METHOD AddIBufferFullChilds
VAR_INPUT
	pFB_ChildTypeIBuffer: POINTER TO FB_IBuffer;
END_VAR
// Method add childs with BufferFull information to the array
IF (usiNumOfIBufferFullChild <= (Base_Const.cMaxNrOfChilds-1)) THEN
	// Add child controller to list
	a_IBufferFullChildCtrl[usiNumOfIBufferFullChild] := pFB_ChildTypeIBuffer^;

	// Inc. number of IBufferFull childs
	usiNumOfIBufferFullChild:= usiNumOfIBufferFullChild+1;
END_IF
END_METHOD

METHOD AddSeqChild
VAR_INPUT
	stSequence: T_Sequence;
END_VAR
// Method add a sequence to list
IF (usiNumOfSeq <= (Base_Const.cMaxNrOfChilds-1)) THEN
	aListOfSeq[usiNumOfSeq].pChild:= stSequence.pChild;
	aListOfSeq[usiNumOfSeq].uinGroupRun:= stSequence.uinGroupRun;
	aListOfSeq[usiNumOfSeq].uinGroupStop:= stSequence.uinGroupStop;
	aListOfSeq[usiNumOfSeq].intCmdSeqRun:= stSequence.intCmdSeqRun;
	aListOfSeq[usiNumOfSeq].intStatusSeqRun:= stSequence.intStatusSeqRun;
	aListOfSeq[usiNumOfSeq].intStatusSeqRun2:= stSequence.intStatusSeqRun2;
	aListOfSeq[usiNumOfSeq].intCmdSeqStop:= stSequence.intCmdSeqStop;
	aListOfSeq[usiNumOfSeq].intStatusSeqStop:= stSequence.intStatusSeqStop;
	// Inc. number of sequence
	usiNumOfSeq:= usiNumOfSeq+1;
	// Check if the pointer is valid
	IF (stSequence.pChild<>0) THEN
		usiNumOfValidPointerSeqChild:= usiNumOfValidPointerSeqChild+1;
	END_IF
END_IF
END_METHOD

METHOD PROTECTED Always : BOOL
SUPER^.Always();

// ---------------------------------------------------------------------------------
// Simulation
IF (CIf.SwCfg.bolSimulation) THEN
	SIf_Cur^.bolKeepAliveHost := NOT SIf_Cur^.bolKeepAlivePlc;
	// Simulate inputs from global module for general supervision (no physical inputs)
	SIf_In^.bolEmoOk.intern := TRUE;
	SIf_In^.bolReady.intern := TRUE;
END_IF

// ----------------------------------------------------------------------------------
// cyclic actions outside of statemachine
IF (me.StateMachine.intState<>cSTA_SINGLE_ANSWER) THEN
	
	// Ready Output
	SIf_Out^.bolReady.intern := (me.StateMachine.intState = BASE_PLC.cSTA_RUN) AND (me.Alarm.eActivAlmClass < BASE_PLC.E_AlmClass.TSTOP);
	
	// Emergency Off
	IF ((SIf_In^.bolEmoOk.intern = FALSE) AND (me.StateMachine.intState <> cSTA_EOFF) AND (me.StateMachine.intState <> cSTA_EOFFBusy)
		AND (me.StateMachine.intState <> cSTA_ERROR) AND (me.StateMachine.intState <> cSTA_ERRORQuit)) THEN
		me.StateMachine.intStateNext := cSTA_EOFFBusy;				
	END_IF
	
	// As long as EMO is not OK, set Alarm
	IF (SIf_In^.bolEmoOk.intern = FALSE) AND ((me.StateMachine.intState = cSTA_EOFF) OR (me.StateMachine.intState = cSTA_EOFFBusy)) THEN
		//SIf_MOD.Alm[E_ALM_MOD.EmergencyOff].strText := 'Emergency off active';
		pfbAlarmCtrl^.setAlarm(CIf.Info.intCtrlId,E_ALM_MOD.EmergencyOff,0,ADR(SIf_MOD.Alm),E_AlmState.RST,CIf.Job.eMe_ActivAlmClass);
	END_IF
	
END_IF

//-------------------------------------------------------------------------------
// Keep Alive function to line controller with togglebit
//-------------------------------------------------------------------------------

// Communication to line control enabled
IF (SIf_Cfg^.bolComToLineControlEnabled = TRUE) THEN
	IF (SIf_Cur^.bolKeepAliveHost <> SIf_Cur^.bolKeepAlivePlc) THEN
		udinTimeToggle_ms := 0;
		SIf_Cur^.bolKeepAlivePlc := SIf_Cur^.bolKeepAliveHost;
	ELSE
		IF (udinTimeToggle_ms >= SIf_Par^.udiComTimeOutLineCtrl_ms) THEN
			//SIf_MOD.Alm[E_ALM_MOD.CommunicationError].strText := 'Communication error to line control'; 
			pfbAlarmCtrl^.setAlarm(CIf.Info.intCtrlId,E_ALM_MOD.CommunicationError,UDINT_TO_DINT(udinTimeToggle_ms),ADR(SIf_MOD.Alm),E_AlmState.RST,CIf.Job.eMe_ActivAlmClass);	
			me.StateMachine.intStateNext := cSTA_Error;	
		END_IF
		udinTimeToggle_ms:= udinTimeToggle_ms + me.FUBInfo.udiSample_ms;
	END_IF
// Communication to line control disabled
ELSE
	SIf_Cur^.bolKeepAliveHost:= NOT SIf_Cur^.bolKeepAlivePlc;
END_IF

//-------------------------------------------------------------------------------
// Calculate the sum of all items in the system and the capacity of the system
//-------------------------------------------------------------------------------
IF (usiNumOfIBufferChild>0) THEN 
	SIf_Cur^.dinNumOfItems:= 0;
	SIf_Cur^.dinMaxCapacity:= 0;
	FOR ii:= 0 TO (usiNumOfIBufferChild-1) DO
		SIf_Cur^.dinNumOfItems:= SIf_Cur^.dinNumOfItems + a_IBufferChildCtrl[ii].NumOfItems;
		SIf_Cur^.dinMaxCapacity:= SIf_Cur^.dinMaxCapacity + a_IBufferChildCtrl[ii].MaxCapacity;
	END_FOR
END_IF

//-------------------------------------------------------------------------------
// Write BufferFull for LineControl into SIF
//-------------------------------------------------------------------------------
IF (usiNumOfIBufferFullChild>0) THEN 
	FOR ii:= 0 TO (usiNumOfIBufferFullChild-1) DO
		SIf_Cur^.a_bBufferIsFull[ii]:= a_IBufferFullChildCtrl[ii].BufferFull;
	END_FOR
END_IF


// ----------------------------------------------------------------------------------
// Conditions Always

// EOFF exist in FB_CtrlModule. Not overrule.
(*
// overrule error always from base -> no EOFF State!! in EOFF go to OFF
IF (me.StateMachine.intStateNext = cSTA_EOFFBusy) THEN
	IF (me.StateMachine.intState=cSTA_OFF) THEN
		me.StateMachine.intStateNext := cSTA_OFF;
	ELSE // stay in OFF
		me.StateMachine.intStateNext := cSTA_OFFBusy;
	END_IF
*)
IF (me.Alarm.eActivAlmClass=E_AlmClass.STOP) AND (me.StateMachine.intStateNext<>cSTA_Error)
		AND ((me.StateMachine.intState = cSTA_RUN) OR (me.StateMachine.intState = cSTA_RUNBusy))THEN
	// alarm evt STOP
	me.StateMachine.intStateNext := cSTA_STOPBusy;	
END_IF
END_METHOD

{attribute 'object_name' := 'CheckAllChildStateOr'}
METHOD PROTECTED CheckAllChildStateOr : BOOL
VAR_INPUT
	In_intCheckState1: INT;
	In_intCheckState2: INT;
END_VAR
VAR
	uinIdx: UINT;
END_VAR
// check if all child controller have reached one of the two In_intCheckState
CheckAllChildStateOr := TRUE;
IF (CIf.Info.uinChildNbr > 0) THEN
	FOR uinIdx := 0 TO CIf.Info.uinChildNbr - 1 DO
		CheckAllChildStateOr := CheckAllChildStateOr AND ((CIf.Info.p_aCIf[uinIdx]^.Job.intState = In_intCheckState1) OR (CIf.Info.p_aCIf[uinIdx]^.Job.intState = In_intCheckState2));
		IF (CheckAllChildStateOr=FALSE) THEN	// at least one child has not whished state reached
			EXIT ;
		END_IF 
	END_FOR
END_IF
END_METHOD

METHOD checkChildAlmClass : BOOL
//------------------------------------------------------------------------------------------------------
// check child alarm classes
// set me alarm class active if at least one child has an EOFF
IF CheckAllChildAlmClass(E_AlmClass.EOFF) THEN
	CIf.Job.eMe_ActivAlmClass := E_AlmClass.EOFF;
	me.Alarm.bolfp := TRUE;
ELSIF CheckAllChildAlmClass(E_AlmClass.OFF) THEN
	CIf.Job.eMe_ActivAlmClass := E_AlmClass.OFF;
	me.Alarm.bolfp := TRUE;
ELSIF CheckAllChildAlmClass(E_AlmClass.STOP) THEN
	CIf.Job.eMe_ActivAlmClass := E_AlmClass.STOP;
	me.Alarm.bolfp := TRUE;
ELSIF CheckAllChildAlmClass(E_AlmClass.TSTOP) THEN
	CIf.Job.eMe_ActivAlmClass := E_AlmClass.TSTOP;
	me.Alarm.bolfp := TRUE;
ELSE
	IF (me.Alarm.bolfp) THEN
		CIf.Job.eMe_ActivAlmClass := E_AlmClass.NONE; // no reset necessary
		me.Alarm.bolfp := FALSE;
	END_IF
END_IF

//------------------------------------------------------------------------------------------------------
// set alarm class parent of childs
//------------------------------------------------------------------------------------------------------
// set alarm class parent of childs in the case of a parent EOFF or me=OFF or EOFF
IF (CIf.Job.eParent_ActivAlmClass=E_AlmClass.EOFF) THEN
	SetAllChildAlmClass(CIf.Job.eParent_ActivAlmClass);
ELSIF(CIf.Job.eMe_ActivAlmClass=E_AlmClass.EOFF) OR (CIf.Job.eMe_ActivAlmClass=E_AlmClass.OFF) THEN
	SetAllChildAlmClass(CIf.Job.eMe_ActivAlmClass);
ELSE
	// no important alarm for child active
	SetAllChildAlmClass(E_AlmClass.NONE);
END_IF
END_METHOD

METHOD PROTECTED checkValidPointer : BOOL
IF (usiNumOfSeq = usiNumOfValidPointerSeqChild) AND (SIf_Cfg<>0) AND (SIf_Par<>0) AND (SIf_Cur<>0) AND (SIf_In<>0) THEN
	checkValidPointer:= TRUE;
ELSE
	// Invalid child pointer
	checkValidPointer:= FALSE;	
	//SIf_MOD.Alm[E_ALM_MOD.InvalidPointer].strText := 'Invalid pointer';
	pfbAlarmCtrl^.setAlarm(CIf.Info.intCtrlId,E_ALM_MOD.InvalidPointer,0,ADR(SIf_MOD.Alm),E_AlmState.RST,CIf.Job.eMe_ActivAlmClass);	
END_IF
END_METHOD

METHOD PUBLIC CtrlInit : BOOL
VAR
	ii: INT;
END_VAR
SUPER^.CtrlInit();

// Initialize all child controller
// Childs are listed in list of sequences
FOR ii:=0 TO usiNumOfSeq-1 BY 1 DO	
	aListOfSeq[ii].pCIF := THIS^.AddChild(aListOfSeq[ii].pChild^);
END_FOR
END_METHOD

METHOD FB_init : BOOL
VAR_INPUT
	///if TRUE, the retain variables are initialized (warm start / cold start)
	bInitRetains: BOOL;
	///if TRUE, the instance afterwards gets moved into the copy code (online change)
	bInCopyCode: BOOL;
END_VAR
VAR
	ii: UINT;
END_VAR
// to manually change in new FUB implementation!!!
// define valid commands for this controller
FOR ii:= 0 TO (SIZEOF(CIf.Job.aCmdList)/SIZEOF(CIf.Job.aCmdList[0])-1) BY 1 DO
	IF (CIf.Job.aCmdList[ii].intCmd=cCMD_INITIALIZED) THEN
		// found first empty array element
		EXIT;
	END_IF
END_FOR

CIf.Job.aCmdList[ii].intCmd := cCMD_RUN;
CIf.Job.aCmdList[ii].strName := 'Run'; 
CIf.Job.aCmdList[ii].bolAvailable := TRUE;
ii := ii +1;
CIf.Job.aCmdList[ii].intCmd := cCMD_STOP;
CIf.Job.aCmdList[ii].strName := 'Stop'; 
CIf.Job.aCmdList[ii].bolAvailable := TRUE;
ii := ii +1;
CIf.Job.aCmdList[ii].intCmd := cCMD_STANDBY;
CIf.Job.aCmdList[ii].strName := 'Standby'; 
CIf.Job.aCmdList[ii].bolAvailable := TRUE;
ii := ii +1;

// set name of class/typ
CIf.Info.strType := 'FB_CtrlModule';
CIf.Info.strFullName := 'Base Controller Module';

// set alarm class
SIf_MOD.Alm[E_ALM_MOD.InvalidPointer].eAlmClass := E_AlmClass.STOP;
SIf_MOD.Alm[E_ALM_MOD.InvalidPointer].strText := 'Invalid pointer';
SIf_MOD.Alm[E_ALM_MOD.CommunicationError].eAlmClass := E_AlmClass.OFF;
SIf_MOD.Alm[E_ALM_MOD.CommunicationError].strText := 'Communication error to line control';
SIf_MOD.Alm[E_ALM_MOD.EmergencyOff].eAlmClass := E_AlmClass.EOFF;
SIf_MOD.Alm[E_ALM_MOD.EmergencyOff].strText := 'Emergency off active';
SIf_MOD.Alm[E_ALM_MOD.TimeoutStartGroup].eAlmClass := E_AlmClass.OFF;
SIf_MOD.Alm[E_ALM_MOD.TimeoutStartGroup].strText := 'Timeout start group';
SIf_MOD.Alm[E_ALM_MOD.TimeoutStopGroup].eAlmClass := E_AlmClass.OFF;
SIf_MOD.Alm[E_ALM_MOD.TimeoutStopGroup].strText := 'Timeout stop group';
SIf_MOD.Alm[E_ALM_MOD.NextModuleNotReadyWarning].eAlmClass := E_AlmClass.WARNING;
SIf_MOD.Alm[E_ALM_MOD.NextModuleNotReadyWarning].strText := 'Next Module is not Ready';
SIf_MOD.Alm[E_ALM_MOD.NextModuleNotReadyStop].eAlmClass := E_AlmClass.STOP;
SIf_MOD.Alm[E_ALM_MOD.NextModuleNotReadyStop].strText := 'Next Module is not Ready';

//*******************************************************************************
// initial values
//*******************************************************************************
udinTimeToggle_ms := 0;
// software configuration
CIf.SwCfg.bolExist := TRUE;
CIf.SwCfg.bolSimulation := FALSE;
me.AlarmConfig.bolChildrenAlarmPropagation := FALSE;

// No initialization for cfg and par in this base module!
// Pointer address of the property is not defined at this time
END_METHOD

METHOD PROTECTED FurtherReactions : BOOL
IF (	(NOT me.AlarmConfig.bolOffAlarmTransitionDisable)	AND (me.Alarm.eActivAlmClass=E_AlmClass.STOP)
	AND (me.StateMachine.intState<>cSTA_ERROR)				AND	(me.StateMachine.intState<>cSTA_ERRORQuit)
	AND	(me.StateMachine.intState<>cSTA_EOFF)				AND	(me.StateMachine.intState<>cSTA_EOFFBusy)
	AND	(me.StateMachine.intState<>cSTA_OFF)				AND	(me.StateMachine.intState<>cSTA_OFFBusy)
	AND (me.StateMachine.intState<>cSTA_STOP)				AND (me.StateMachine.intState<>cSTA_STOPBusy)
	AND	(me.StateMachine.intState>cSTA_PON)) THEN
	
	me.StateMachine.intStateNext := cSTA_STOPBusy;
	me.StateMachine.intState := cSTA_DONE;
	
ELSIF (	(NOT me.AlarmConfig.bolOffAlarmTransitionDisable)	AND (me.Alarm.eActivAlmClass=E_AlmClass.TSTOP)
	AND (me.StateMachine.intState<>cSTA_ERROR)				AND	(me.StateMachine.intState<>cSTA_ERRORQuit)
	AND	(me.StateMachine.intState<>cSTA_EOFF)				AND	(me.StateMachine.intState<>cSTA_EOFFBusy)
	AND	(me.StateMachine.intState<>cSTA_OFF)				AND	(me.StateMachine.intState<>cSTA_OFFBusy)
	AND (me.StateMachine.intState<>cSTA_STOP)				AND (me.StateMachine.intState<>cSTA_STOPBusy)
	AND	(me.StateMachine.intState>cSTA_PON)) THEN
	
	me.StateMachine.intStateNext := cSTA_STOPBusy;
	me.StateMachine.intState := cSTA_DONE;
	
END_IF
END_METHOD

METHOD PROTECTED getCmdState : STRING
VAR_INPUT
	intCmdState: INT;
	bolState: BOOL;
END_VAR
getCmdState := SUPER^.getCmdState(intCmdState:=intCmdState,bolState:=bolState); // get global/base defined cmds/states
IF (getCmdState='') THEN // global not defined get local
	// get string cmd/state string information in runtime
	IF (bolState=FALSE) THEN
		// cmd's
		CASE intCmdState OF
			cCMD_STANDBY: 
				getCmdState := 'cCMD_STANDBY';
		END_CASE
	ELSE
		// states
		CASE intCmdState OF	
			cSTA_STANDBY:
				getCmdState := 'cSTA_STANDBY';
			cSTA_STANDBYBusy:
				getCmdState := 'cSTA_STANDBYBusy';
			// SUB States
			cSTA_SUB_INITIALIZED:
				getCmdState := 'cSTA_SUB_INITIALIZED';
			cSTA_SUB_SEND_GROUP_CMD:
				getCmdState := 'cSTA_SUB_SEND_GROUP_CMD';
			cSTA_SUB_CHECK_GROUP_STATUS:
				getCmdState := 'cSTA_SUB_CHECK_GROUP_STATUS';
			cSTA_SUB_WAIT:
				getCmdState := 'cSTA_SUB_WAIT';
			cSTA_SUB_FINISHED:
				getCmdState := 'cSTA_SUB_FINISHED';
		END_CASE;
	END_IF
END_IF
END_METHOD

METHOD PROTECTED IoInBridge : BOOL
// digitale and analoge inputs read from hardware or forcing
SIf_In^.bolReady.map	:= THIS^.In_bolReady;
SIf_In^.bolEmoOk.map	:= THIS^.In_bolEmoOk;

IF (CIf.SwCfg.bolSimulation = FALSE) THEN
	BASE_PLC.getInBol(CIf.Job.bolIoForce,ADR(SIf_In^.bolReady));
	BASE_PLC.getInBol(CIf.Job.bolIoForce,ADR(SIf_In^.bolEmoOk));
ELSE
	//simulation of global IO
	SIf_In^.bolReady.intern	:= TRUE;
	SIf_In^.bolEmoOk.intern	:= TRUE;
END_IF
END_METHOD

METHOD PROTECTED IoOutBridge : BOOL
// digitale and analoge inputs read from hardware or forcing
IF (CIf.SwCfg.bolSimulation = FALSE) THEN
	
	setOutBol(CIf.Job.bolIoForce ,ADR(SIf_Out^.bolReady));
	THIS^.Out_bolReady := SIf_Out^.bolReady.map;

	// check interlocks to prevent damages
	IF (CIf.Job.bolIlkOverwrite=FALSE) THEN
	;
	END_IF
END_IF
END_METHOD

PROPERTY SIf_Cfg : POINTER TO T_Ctrl_SIf_MOD_Cfg
GET
SIf_Cfg:= SIf_MOD.Cfg;
END_GET
SET
SIf_MOD.Cfg := SIf_Cfg;
END_SET
END_PROPERTY

PROPERTY SIf_Cur : POINTER TO T_Ctrl_SIf_MOD_Cur
GET
SIf_Cur:= SIf_MOD.Cur;
END_GET
SET
SIf_MOD.Cur := SIf_Cur;
END_SET
END_PROPERTY

PROPERTY SIf_In : POINTER TO T_Ctrl_SIf_MOD_In
GET
SIf_In:= SIf_MOD.In;
END_GET
SET
SIf_MOD.In := SIf_In;
END_SET
END_PROPERTY

PROPERTY SIf_Out : POINTER TO T_Ctrl_SIf_MOD_Out
GET
SIf_Out:= SIf_MOD.Out;
END_GET
SET
SIf_MOD.Out := SIf_Out;
END_SET
END_PROPERTY

PROPERTY SIf_Par : POINTER TO T_Ctrl_SIf_MOD_Par
GET
SIf_Par:= SIf_MOD.Par;
END_GET
SET
SIf_MOD.Par := SIf_Par;
END_SET
END_PROPERTY

METHOD PROTECTED sta_EOFF : BOOL
// state implemetation
//--------------------------------------------------------------------------------------
// Entry action
	IF (me.StateMachine.intState<>me.StateMachine.intStateLastCycle) THEN
		me.StateMachine.intStateLastCycle := me.StateMachine.intState;	
	END_IF

//--------------------------------------------------------------------------------------
// Cyclic action
	IF (me.StateMachine.intState=me.StateMachine.intStateLastCycle) THEN		
		
		// As long as the EMO is not reseted!
		IF NOT (SIf_In^.bolEmoOk.intern) THEN
			// Clear pending and new commands cyclic to prevent automatic recovery!
			CIf.Job.intACmd := BASE_PLC.cCMD_DONE;
			CIf.Job.intMCmd := BASE_PLC.cCMD_DONE;
		END_IF
	
		// State Change Condition
		IF (SIf_In^.bolEmoOk.intern) AND (me.Alarm.eActivAlmClass<>E_AlmClass.EOFF) AND (me.intCmd<>BASE_PLC.cCMD_EOFF) AND (me.intCmd<>BASE_PLC.cCMD_DONE) THEN
			me.StateMachine.intStateNext := cSTA_OFF;
		END_IF
	END_IF

//--------------------------------------------------------------------------------------
// Exit action
	IF (me.StateMachine.intState<>me.StateMachine.intStateNext) THEN
		;
	END_IF
END_METHOD

METHOD PROTECTED sta_EOFFBusy : BOOL
// state implemetation
//--------------------------------------------------------------------------------------
// Entry action
	IF (me.StateMachine.intState<>me.StateMachine.intStateLastCycle) THEN
		me.StateMachine.intStateLastCycle := me.StateMachine.intState;
	END_IF

	
//--------------------------------------------------------------------------------------
// Cyclic action
	IF (me.StateMachine.intState=me.StateMachine.intStateLastCycle) THEN
		
		// In case of an emergency, set all childs to off 
		// Set in cyclic action because of possible errors or manual/auto changes!
		SUPER^.SetAllChildCmd(BASE_PLC.cCMD_OFF);

		// check if all childs have reached the state
		IF CheckAllChildState(cSTA_OFF) THEN
			me.StateMachine.intStateNext := cSTA_EOFF;
		END_IF
	END_IF

	
//--------------------------------------------------------------------------------------
// Exit action
	IF (me.StateMachine.intState<>me.StateMachine.intStateNext) THEN
		;
	END_IF
END_METHOD

METHOD PROTECTED sta_ERROR : BOOL
// state implemetation
//--------------------------------------------------------------------------------------
// Entry action
	IF (me.StateMachine.intState<>me.StateMachine.intStateLastCycle) THEN
		me.StateMachine.intStateHistory := me.StateMachine.intStateLastCycle; // -> possibillity to go back to state before error
		me.StateMachine.intStateLastCycle := me.StateMachine.intState;
		// Clear pending command to prevent automatic recovery!
		CIf.Job.intACmd:=cSTA_DONE;
		// In case on an error, set all childs to off
		SetAllChildCmd(cCMD_OFF);
	END_IF

//--------------------------------------------------------------------------------------
// Cyclic action
	IF (me.StateMachine.intState=me.StateMachine.intStateLastCycle) THEN
		
		;
		// State Change Condition
		IF ((CIf.Job.bolAlmReset = TRUE) AND (CheckAllChildState(cSTA_OFF))) THEN
			me.StateMachine.intStateNext := cSTA_ERRORQuit;
		END_IF
	END_IF

//--------------------------------------------------------------------------------------
// Exit action
	IF (me.StateMachine.intState<>me.StateMachine.intStateNext) THEN
		;
	END_IF
END_METHOD

METHOD PROTECTED sta_OFF : BOOL
// state implemetation
//--------------------------------------------------------------------------------------
// Entry action
	IF (me.StateMachine.intState<>me.StateMachine.intStateLastCycle) THEN
		me.StateMachine.intStateLastCycle := me.StateMachine.intState;
	END_IF

	
//--------------------------------------------------------------------------------------
// Cyclic action
	IF (me.StateMachine.intState=me.StateMachine.intStateLastCycle) THEN
				
		// State Change Condition
		IF (me.Alarm.eActivAlmClass < E_AlmClass.TSTOP) THEN
			IF (me.intCmd=cCMD_RUN) THEN
				IF (SIf_In^.bolReady.intern OR SIf_Cfg^.bolIgnoreReadyInput) THEN 
					me.StateMachine.intStateNext := cSTA_RUNBusy;
				ELSE
					//SIf_MOD.Alm[E_ALM_MOD.NextModuleNotReadyWarning].strText := 'Next Module is not Ready';
					pfbAlarmCtrl^.setAlarm(CIf.Info.intCtrlId,E_ALM_MOD.NextModuleNotReadyWarning,0,ADR(SIf_MOD.Alm),E_AlmState.RST,CIf.Job.eMe_ActivAlmClass);
					CIf.Job.intACmd := cCMD_DONE;
				END_IF
			END_IF
		END_IF
	END_IF

	
//--------------------------------------------------------------------------------------
// Exit action
	IF (me.StateMachine.intState<>me.StateMachine.intStateNext) THEN
		;
	END_IF
END_METHOD

METHOD PROTECTED sta_OFFBusy : BOOL
// state implemetation
//--------------------------------------------------------------------------------------
// Entry action
	IF (me.StateMachine.intState<>me.StateMachine.intStateLastCycle) THEN
		me.StateMachine.intStateLastCycle := me.StateMachine.intState;
		
		// Set commandos not only in entry action because of possible errors or manual/auto changes
		// PRE/AVME 06.01.2014
		//SetAllChildCmd(cCMD_OFF); // set acmd off all childs 
	END_IF


//--------------------------------------------------------------------------------------
// Cyclic action
	IF (me.StateMachine.intState=me.StateMachine.intStateLastCycle) THEN
		
		SetAllChildCmd(cCMD_OFF); // set acmd off all childs 
		
		// State Change Condition
		IF (CheckAllChildState(cSTA_OFF)) THEN
			me.StateMachine.intStateNext := cSTA_OFF;
		ELSIF (me.intCmd=cCMD_RUN) AND (me.Alarm.eActivAlmClass < E_AlmClass.TSTOP) THEN
			me.StateMachine.intStateNext := cSTA_RUNBusy;
		END_IF
	END_IF


//--------------------------------------------------------------------------------------
// Exit action
	IF (me.StateMachine.intState<>me.StateMachine.intStateNext) THEN
		;
	END_IF
END_METHOD

{attribute 'object_name' := 'sta_PONBusy'}
METHOD PROTECTED sta_PONBusy : BOOL
// state implemetation
//--------------------------------------------------------------------------------------
// Entry action
	IF (me.StateMachine.intState<>me.StateMachine.intStateLastCycle) THEN
		me.StateMachine.intStateLastCycle := me.StateMachine.intState;
		
		SetAllChildCmd(cCMD_PON); // set acmd off all childs 
	END_IF


//--------------------------------------------------------------------------------------
// Cyclic action
	IF (me.StateMachine.intState=me.StateMachine.intStateLastCycle) THEN

		// State Change Condition
		IF (FALSE) THEN
			;
		ELSIF CheckAllChildStateOr(cSTA_PON, cSTA_RUN) THEN
			me.StateMachine.intStateNext := cSTA_PON;
		END_IF
		
	END_IF


//--------------------------------------------------------------------------------------
// Exit action
	IF (me.StateMachine.intState<>me.StateMachine.intStateNext) THEN
		;
	END_IF
END_METHOD

METHOD PROTECTED sta_RUN : BOOL
// state implemetation
//--------------------------------------------------------------------------------------
// Entry action
	IF (me.StateMachine.intState<>me.StateMachine.intStateLastCycle) THEN
		me.StateMachine.intStateLastCycle := me.StateMachine.intState;
		;
	END_IF

//--------------------------------------------------------------------------------------
// Cyclic action
	IF (me.StateMachine.intState=me.StateMachine.intStateLastCycle) THEN

		// Simulation
		IF (CIf.SwCfg.bolSimulation) THEN
			;
		END_IF

		// State Change Condition	
		IF (me.intCmd=cCMD_STOP) THEN
			me.StateMachine.intStateNext :=  cSTA_STOPBusy;
		ELSIF NOT (SIf_In^.bolReady.intern OR SIf_Cfg^.bolIgnoreReadyInput) THEN
			//SIf_MOD.Alm[E_ALM_MOD.NextModuleNotReadyStop].strText := 'Next Module is not Ready';
			pfbAlarmCtrl^.setAlarm(CIf.Info.intCtrlId,E_ALM_MOD.NextModuleNotReadyStop,0,ADR(SIf_MOD.Alm),E_AlmState.RST,CIf.Job.eMe_ActivAlmClass);
			me.StateMachine.intStateNext := cSTA_STOPBusy;
			CIf.Job.intACmd := cCMD_DONE;
		END_IF

	END_IF

//--------------------------------------------------------------------------------------
// Exit action
	IF (me.StateMachine.intState<>me.StateMachine.intStateNext) THEN
		;
	END_IF
END_METHOD

METHOD PROTECTED sta_RUNBusy : BOOL
VAR
	ii: INT;
	bolFurtherGrpExist: BOOL;
END_VAR
// state implemetation
//--------------------------------------------------------------------------------------
// Entry action
	IF (me.StateMachine.intState<>me.StateMachine.intStateLastCycle) THEN
		me.StateMachine.intStateLastCycle := me.StateMachine.intState;
		// Init sub state machine
		me.SubStateMachine.intState := cSTA_SUB_INITIALIZED; 
		me.SubStateMachine.intStateNext := cSTA_SUB_INITIALIZED;
	END_IF

//--------------------------------------------------------------------------------------
// Cyclic action
	IF (me.StateMachine.intState=me.StateMachine.intStateLastCycle) THEN

		// Simulation
		IF (CIf.SwCfg.bolSimulation) THEN
			;
		END_IF
	
		// Start Cycle with substates	
		//--------------------------------------------------------------------------------------
		// sub state machine for sequence
		CASE me.SubStateMachine.intState OF
			//--------------------------------------------------------------------------------------
			cSTA_SUB_INITIALIZED:
			
				// Loop over all registered childs
				FOR ii:=0 TO usiNumOfSeq-1 BY 1 DO
					// Clear checked flag		
					aListOfSeq[ii].bolChecked:= FALSE;
				END_FOR
				uinGroupIndex:= 1;
				me.SubStateMachine.intStateNext := cSTA_SUB_SEND_GROUP_CMD;
				
			cSTA_SUB_SEND_GROUP_CMD:
				
				intCheckCounter:= 0;
				// Loop over all registered childs
				FOR ii:=0 TO usiNumOfSeq-1 BY 1 DO
					// If child is associated for the current group index		
					IF (aListOfSeq[ii].uinGroupRun = uinGroupIndex) THEN
						// Send defined command
						aListOfSeq[ii].pCIF^.Job.intACmd:= aListOfSeq[ii].intCmdSeqRun;
						intCheckCounter:= intCheckCounter + 1;
					END_IF			
				END_FOR
				// Change state
				me.SubStateMachine.intStateNext := cSTA_SUB_CHECK_GROUP_STATUS;
			
			
			cSTA_SUB_CHECK_GROUP_STATUS:
	
				// Loop over all registered childs
				FOR ii:=0 TO usiNumOfSeq-1 BY 1 DO
					// If child is associated for the current group index		
					IF (aListOfSeq[ii].uinGroupRun = uinGroupIndex) THEN
						// Check defined status and if child not already checked
						IF (((aListOfSeq[ii].pCIF^.Job.intState = aListOfSeq[ii].intStatusSeqRun) OR 
						(aListOfSeq[ii].pCIF^.Job.intState = aListOfSeq[ii].intStatusSeqRun2)) AND (aListOfSeq[ii].bolChecked = FALSE)) THEN
							aListOfSeq[ii].bolChecked:= TRUE;
							intCheckCounter:= intCheckCounter - 1;
						END_IF				
					END_IF			
				END_FOR
				
				// All childs in group has the right state
				IF (intCheckCounter <= 0) THEN		
					bolFurtherGrpExist:= FALSE;
					// Check if a further group exist!	
					FOR ii:=0 TO usiNumOfSeq-1 BY 1 DO	
						IF (aListOfSeq[ii].uinGroupRun > uinGroupIndex) THEN
							bolFurtherGrpExist:= TRUE;
							EXIT;
						END_IF			
					END_FOR
					// further group exist
					IF (bolFurtherGrpExist = TRUE) THEN
						IF (uinGroupIndex < uinMaxNrOfGroups) THEN			
							me.SubStateMachine.intStateNext := cSTA_SUB_WAIT;	
						END_IF
					ELSE
						me.SubStateMachine.intStateNext := cSTA_SUB_FINISHED;		
					END_IF
				END_IF

			cSTA_SUB_WAIT:
				
				IF (me.SubStateMachine.udiTimeInState_ms >= SIf_Par^.aListOfRunGrpWaitTime_ms[uinGroupIndex-1]) THEN
					// Inc. group index 
					uinGroupIndex:= uinGroupIndex + 1;	
					// Change state, send command for next group
					me.SubStateMachine.intStateNext := cSTA_SUB_SEND_GROUP_CMD;
				END_IF
			
			cSTA_SUB_FINISHED:
					;		
		END_CASE
		
		// Check time out error
		IF (SIf_MOD.Par^.udiTimeoutStarting_ms <> 0) AND (me.SubStateMachine.udiTimeInState_ms > (SIf_Par^.aListOfRunGrpWaitTime_ms[uinGroupIndex-1] + SIf_MOD.Par^.udiTimeoutStarting_ms)) THEN
			//SIf_MOD.Alm[E_ALM_MOD.TimeoutStarGroup].strText := 'Timeout start group';
			pfbAlarmCtrl^.setAlarm(CIf.Info.intCtrlId,E_ALM_MOD.TimeoutStartGroup,uinGroupIndex,ADR(SIf_MOD.Alm),E_AlmState.RST,CIf.Job.eMe_ActivAlmClass);
			me.StateMachine.intStateNext := cSTA_ERROR;
		END_IF
		
		// State Change Condition
		IF (me.intCmd=cCMD_STOP) THEN
			me.StateMachine.intStateNext :=  cSTA_STOPBusy;
		ELSIF NOT (SIf_In^.bolReady.intern OR SIf_Cfg^.bolIgnoreReadyInput) THEN
			//SIf_MOD.Alm[E_ALM_MOD.NextModuleNotReadyStop].strText := 'Next Module is not Ready';
			pfbAlarmCtrl^.setAlarm(CIf.Info.intCtrlId,E_ALM_MOD.NextModuleNotReadyStop,0,ADR(SIf_MOD.Alm),E_AlmState.RST,CIf.Job.eMe_ActivAlmClass);
			me.StateMachine.intStateNext := cSTA_STOPBusy;
			CIf.Job.intACmd := cCMD_DONE;
		ELSIF (me.SubStateMachine.intState = cSTA_SUB_FINISHED) THEN
			me.StateMachine.intStateNext := cSTA_RUN;
		END_IF
	END_IF

//--------------------------------------------------------------------------------------
// Exit action
	IF (me.StateMachine.intState<>me.StateMachine.intStateNext) THEN
		;
	END_IF
END_METHOD

METHOD PROTECTED sta_STANDBY : BOOL
// state implemetation
//--------------------------------------------------------------------------------------
// Entry action
	IF (me.StateMachine.intState<>me.StateMachine.intStateLastCycle) THEN
		me.StateMachine.intStateLastCycle := me.StateMachine.intState;
	END_IF

	
//--------------------------------------------------------------------------------------
// Cyclic action
	IF (me.StateMachine.intState=me.StateMachine.intStateLastCycle) THEN
		
		// State Change Condition	
		IF (me.intCmd=cCMD_STOP) THEN
			me.StateMachine.intStateNext :=  cSTA_STOPBusy;
		ELSIF NOT (SIf_In^.bolReady.intern OR SIf_Cfg^.bolIgnoreReadyInput) THEN
			//SIf_MOD.Alm[E_ALM_MOD.NextModuleNotReadyStop].strText := 'Next Module is not Ready';
			pfbAlarmCtrl^.setAlarm(CIf.Info.intCtrlId,E_ALM_MOD.NextModuleNotReadyStop,0,ADR(SIf_MOD.Alm),E_AlmState.RST,CIf.Job.eMe_ActivAlmClass);
			me.StateMachine.intStateNext := cSTA_STOPBusy;
			CIf.Job.intACmd := cCMD_DONE;
		ELSIF (me.intCmd=cCMD_RUN) THEN
			me.StateMachine.intStateNext :=  cSTA_RUNBusy;
		END_IF
		
	END_IF

	
//--------------------------------------------------------------------------------------
// Exit action
	IF (me.StateMachine.intState<>me.StateMachine.intStateNext) THEN
		;
	END_IF
END_METHOD

METHOD PROTECTED sta_STANDBYBusy : BOOL
// state implemetation
//--------------------------------------------------------------------------------------
// Entry action
	IF (me.StateMachine.intState<>me.StateMachine.intStateLastCycle) THEN
		me.StateMachine.intStateLastCycle := me.StateMachine.intState;
	END_IF


//--------------------------------------------------------------------------------------
// Cyclic action
	IF (me.StateMachine.intState=me.StateMachine.intStateLastCycle) THEN
		
		// State Change Condition	
		IF (me.intCmd=cCMD_STOP) THEN
			me.StateMachine.intStateNext :=  cSTA_STOPBusy;
		ELSIF NOT (SIf_In^.bolReady.intern OR SIf_Cfg^.bolIgnoreReadyInput) THEN
			//SIf_MOD.Alm[E_ALM_MOD.NextModuleNotReadyStop].strText := 'Next Module is not Ready';
			pfbAlarmCtrl^.setAlarm(CIf.Info.intCtrlId,E_ALM_MOD.NextModuleNotReadyStop,0,ADR(SIf_MOD.Alm),E_AlmState.RST,CIf.Job.eMe_ActivAlmClass);
			me.StateMachine.intStateNext := cSTA_STOPBusy;
			CIf.Job.intACmd := cCMD_DONE;
		ELSIF (me.intCmd=cCMD_RUN) THEN
			me.StateMachine.intStateNext :=  cSTA_RUNBusy;
		ELSE
			me.StateMachine.intStateNext :=  cSTA_STANDBY;
		END_IF
		
	END_IF


//--------------------------------------------------------------------------------------
// Exit action
	IF (me.StateMachine.intState<>me.StateMachine.intStateNext) THEN
		;
	END_IF
END_METHOD

METHOD PROTECTED sta_STOP : BOOL
// state implemetation
//--------------------------------------------------------------------------------------
// Entry action
	IF (me.StateMachine.intState<>me.StateMachine.intStateLastCycle) THEN
		me.StateMachine.intStateLastCycle := me.StateMachine.intState;
	END_IF


//--------------------------------------------------------------------------------------
// Cyclic action
	IF (me.StateMachine.intState=me.StateMachine.intStateLastCycle) THEN
		
		// State Change Condition
		IF (me.Alarm.eActivAlmClass<E_AlmClass.TSTOP) THEN
			IF (me.intCmd=cCMD_RUN) THEN
				IF (SIf_In^.bolReady.intern OR SIf_Cfg^.bolIgnoreReadyInput) THEN 
					me.StateMachine.intStateNext := cSTA_RUNBusy;
				ELSE
					//SIf_MOD.Alm[E_ALM_MOD.NextModuleNotReadyWarning].strText := 'Next Module is not Ready';
					pfbAlarmCtrl^.setAlarm(CIf.Info.intCtrlId,E_ALM_MOD.NextModuleNotReadyWarning,0,ADR(SIf_MOD.Alm),E_AlmState.RST,CIf.Job.eMe_ActivAlmClass);
					CIf.Job.intACmd := cCMD_DONE;
				END_IF
			END_IF
		END_IF
	END_IF

//--------------------------------------------------------------------------------------
// Exit action
	IF (me.StateMachine.intState<>me.StateMachine.intStateNext) THEN
		;
	END_IF
END_METHOD

METHOD PROTECTED sta_STOPBusy : BOOL
VAR
	ii: INT;
	bolFurtherGrpExist: BOOL;
END_VAR
// state implemetation
//--------------------------------------------------------------------------------------
// Entry action
	IF (me.StateMachine.intState<>me.StateMachine.intStateLastCycle) THEN
		me.StateMachine.intStateLastCycle := me.StateMachine.intState;	
		// Init sub state machine
		me.SubStateMachine.intState := cSTA_SUB_INITIALIZED; 
		me.SubStateMachine.intStateNext := cSTA_SUB_INITIALIZED;
	END_IF


//--------------------------------------------------------------------------------------
// Cyclic action
	IF (me.StateMachine.intState=me.StateMachine.intStateLastCycle) THEN

		// Simulation
		IF (CIf.SwCfg.bolSimulation) THEN
			;
		END_IF
		
		// Stop Cycle with substates	
		//--------------------------------------------------------------------------------------
		// sub state machine for sequence
		CASE me.SubStateMachine.intState OF
			//--------------------------------------------------------------------------------------
			cSTA_SUB_INITIALIZED:
			
				// Loop over all registered childs
				FOR ii:=0 TO usiNumOfSeq-1 BY 1 DO
					// Clear checked flag		
					aListOfSeq[ii].bolChecked:= FALSE;
				END_FOR
				uinGroupIndex:= 1;
				me.SubStateMachine.intStateNext := cSTA_SUB_SEND_GROUP_CMD;
				
			cSTA_SUB_SEND_GROUP_CMD:
				
				intCheckCounter:= 0;
				// Loop over all registered childs
				FOR ii:=0 TO usiNumOfSeq-1 BY 1 DO
					// If child is associated for the current group index		
					IF (aListOfSeq[ii].uinGroupStop = uinGroupIndex) THEN
						// Send defined command
						aListOfSeq[ii].pCIF^.Job.intACmd:= aListOfSeq[ii].intCmdSeqStop;
						intCheckCounter:= intCheckCounter + 1;
					END_IF			
				END_FOR
				// Change state
				me.SubStateMachine.intStateNext := cSTA_SUB_CHECK_GROUP_STATUS;
			
			
			cSTA_SUB_CHECK_GROUP_STATUS:
	
				// Loop over all registered childs
				FOR ii:=0 TO usiNumOfSeq-1 BY 1 DO
					// If child is associated for the current group index		
					IF (aListOfSeq[ii].uinGroupStop = uinGroupIndex) THEN
						// Check defined status and if child not already checked
						IF ((aListOfSeq[ii].pCIF^.Job.intState = aListOfSeq[ii].intStatusSeqStop) AND (aListOfSeq[ii].bolChecked = FALSE)) THEN
							aListOfSeq[ii].bolChecked:= TRUE;
							intCheckCounter:= intCheckCounter - 1;
						END_IF				
					END_IF			
				END_FOR
				
				// All childs in group has the right state
				IF (intCheckCounter <= 0) THEN		
					bolFurtherGrpExist:= FALSE;
					// Check if a further group exist!	
					FOR ii:=0 TO usiNumOfSeq-1 BY 1 DO	
						IF (aListOfSeq[ii].uinGroupStop > uinGroupIndex) THEN
							bolFurtherGrpExist:= TRUE;
							EXIT;
						END_IF			
					END_FOR
					// further group exist
					IF (bolFurtherGrpExist = TRUE) THEN
						IF (uinGroupIndex < uinMaxNrOfGroups) THEN			
							me.SubStateMachine.intStateNext := cSTA_SUB_WAIT;	
						END_IF
					ELSE
						me.SubStateMachine.intStateNext := cSTA_SUB_FINISHED;		
					END_IF
				END_IF

			cSTA_SUB_WAIT:
				
				IF (me.SubStateMachine.udiTimeInState_ms >= SIf_Par^.aListOfStopGrpWaitTime_ms[uinGroupIndex-1]) THEN
					// Inc. group index 
					uinGroupIndex:= uinGroupIndex + 1;	
					// Change state, send command for next group
					me.SubStateMachine.intStateNext := cSTA_SUB_SEND_GROUP_CMD;
				END_IF
			
			cSTA_SUB_FINISHED:
					;		
		END_CASE
		
		// Check time out error
		IF (SIf_MOD.Par^.udiTimeoutStopping_ms <> 0) AND (me.SubStateMachine.udiTimeInState_ms > (SIf_Par^.aListOfStopGrpWaitTime_ms[uinGroupIndex-1] + SIf_MOD.Par^.udiTimeoutStopping_ms)) THEN
			//SIf_MOD.Alm[E_ALM_MOD.TimeoutStopGroup].strText := 'Timeout stop group';
			pfbAlarmCtrl^.setAlarm(CIf.Info.intCtrlId,E_ALM_MOD.TimeoutStopGroup,uinGroupIndex,ADR(SIf_MOD.Alm),E_AlmState.RST,CIf.Job.eMe_ActivAlmClass);
			me.StateMachine.intStateNext := cSTA_ERROR;
		END_IF
	
		// State Change Condition
		IF (me.SubStateMachine.intState = cSTA_SUB_FINISHED) THEN
			me.StateMachine.intStateNext := cSTA_STOP;
		ELSIF (me.intCmd=cCMD_RUN) THEN
			// State Change Condition
			IF (me.Alarm.eActivAlmClass<E_AlmClass.TSTOP) THEN	
				me.StateMachine.intStateNext := cSTA_RUNBusy;	
			ELSE
				// Clear pending command to prevent automatic recovery!
				CIf.Job.intACmd:=cSTA_DONE;
			END_IF
		END_IF

	END_IF

//--------------------------------------------------------------------------------------
// Exit action
	IF (me.StateMachine.intState<>me.StateMachine.intStateNext) THEN
		;
	END_IF
END_METHOD

METHOD PROTECTED StateMachine : BOOL
SUPER^.StateMachine();

// main statemachine of base controller
CASE me.StateMachine.intState OF
	cSTA_RUN: 
        THIS^.sta_RUN();
    cSTA_RUNBusy: 
        THIS^.sta_RUNBusy();
	cSTA_STOP: 
        THIS^.sta_STOP();
    cSTA_STOPBusy: 
        THIS^.sta_STOPBusy();
	cSTA_STANDBY:
		THIS^.sta_STANDBY();
	cSTA_STANDBYBusy:
		THIS^.sta_STANDBYBusy();
END_CASE;
END_METHOD

END_FUNCTION_BLOCK

// POUs/Controller/Lvl3/BaseCtrlModule/IBuffer
INTERFACE IBuffer

PROPERTY BufferFull : BOOL
GET
END_GET
END_PROPERTY

PROPERTY MaxCapacity : DINT
GET
END_GET
END_PROPERTY

PROPERTY NumOfItems : DINT
GET
END_GET
END_PROPERTY

END_INTERFACE

// POUs/Controller/Lvl3/BaseCtrlModule/FB_IBuffer
///FUNCTION_BLOCK PUBLIC FB_IBuffer IMPLEMENTS IBuffer
FUNCTION_BLOCK FB_IBuffer EXTENDS FB_CtrlBase IMPLEMENTS IBuffer

// This is a Dummy-FB, used for the interface (IBuffer) to the buffer-modules

PROPERTY BufferFull : BOOL
GET
END_GET
END_PROPERTY

PROPERTY MaxCapacity : DINT
GET
END_GET
END_PROPERTY

PROPERTY NumOfItems : DINT
GET
END_GET
END_PROPERTY

END_FUNCTION_BLOCK

// POUs/Utility/AFF [Array Fifo]/FB_ArrayFifo
FUNCTION_BLOCK FB_ArrayFifo
VAR
	/// Internal buffer
	m_pItemBuffer: POINTER TO BYTE;
	m_uinItemSize: UINT;
	/// Actual Count of the elements in the buffer
	m_uinItemCount: UINT;
	/// Index of the first added element
	m_iFirstElement: INT;
	/// Index of the last added element
	m_iLastElement: INT;
	m_uinBufferSize: UINT := 0;
	m_uinMaxItemCount: UINT := 0;
	m_bolFreePointer: BOOL := FALSE;
	fbFifo: Tc2_Utilities.FB_MemRingBuffer;
END_VAR

PROPERTY FreePointer : BOOL
GET
FreePointer := m_bolFreePointer;
END_GET
SET
m_bolFreePointer := FreePointer;
END_SET
END_PROPERTY

{attribute 'object_name' := 'Initialize'}
METHOD Initialize : BOOL
VAR_INPUT
	/// Size of one item [byte]
	uinItemSize: UINT;
	/// Buffer for the items to be stored in.
	pBuffer: POINTER TO BYTE;
	/// Buffer Size in [byte]
	uinBufferSize: UINT;
END_VAR
Initialize := FALSE;

IF (pBuffer <> Tc3_MemMan.NULL) AND (uinItemSize > 0) AND (uinBufferSize > 0) THEN
	m_pItemBuffer := pBuffer;
	m_uinBufferSize := uinBufferSize;
	m_uinItemSize := uinItemSize;
	m_uinMaxItemCount := uinBufferSize / uinItemSize;
	
	fbFifo.cbBuffer 	:= uinBufferSize;
	fbFifo.pBuffer  	:= pBuffer;
	
	Initialize := TRUE;
END_IF
END_METHOD

PROPERTY ItemCount : UINT
GET
ItemCount := UDINT_TO_UINT(fbFifo.nCount);
END_GET
END_PROPERTY

PROPERTY MaxBufferSize : INT
GET
MaxBufferSize := UINT_TO_INT(m_uinBufferSize);
END_GET
END_PROPERTY

{attribute 'object_name' := 'Peek'}
METHOD Peek : BOOL
VAR_INPUT
	pData: POINTER TO BYTE;
END_VAR
Peek := FALSE;

IF fbFifo.nCount > 0 THEN
	fbFifo.cbRead := m_uinItemSize;
	fbFifo.pRead := pData;
	fbFifo.A_GetHead();
	
	Peek := fbFifo.bOk;
END_IF
END_METHOD

{attribute 'object_name' := 'Pop'}
METHOD Pop : BOOL
VAR_INPUT
	pData: POINTER TO BYTE;
END_VAR
Pop := FALSE;

IF fbFifo.nCount > 0 THEN
	fbFifo.cbRead := m_uinItemSize;
	fbFifo.pRead := pData;
	fbFifo.A_RemoveHead();
	m_uinItemCount := UDINT_TO_UINT(fbFifo.nCount);
	
	Pop := fbFifo.bOk;
END_IF
END_METHOD

{attribute 'object_name' := 'Push'}
METHOD Push : INT
VAR_INPUT
	pData: POINTER TO BYTE;
END_VAR
Push := -1;

IF fbFifo.nCount < m_uinBufferSize THEN
	fbFifo.cbWrite := m_uinItemSize;
	fbFifo.pWrite  := pData;
	fbFifo.A_AddTail();
	m_uinItemCount := UDINT_TO_UINT(fbFifo.nCount);

	IF fbFifo.bOk THEN
		IF m_bolFreePointer THEN
			__DELETE(pData);
		END_IF
		
		Push := UINT_TO_INT(m_uinItemCount);
	END_IF
END_IF
END_METHOD

ACTION Reset:
fbFifo.A_Reset();
m_uinItemCount := 0;
END_ACTION

END_FUNCTION_BLOCK

// POUs/Utility/CFR [Csv File Reader]/FB_CFR
FUNCTION_BLOCK FB_CFR
VAR_INPUT
	sFileName	: T_MaxString; (* CSV source file path and name *)
	bRead		: BOOL			:= FALSE; (* Rising edge starts program execution *)
END_VAR
VAR_OUTPUT
	bBusy		: BOOL;
	values	: ARRAY[0..MAX_CSV_ROWS-1, 0..MAX_CSV_COLUMNS-1] OF STRING(MAX_CSV_FIELD_LENGTH); (* Target PLC database *)
END_VAR
VAR CONSTANT
	MAX_CSV_ROWS 			: UINT := 100;
	MAX_CSV_COLUMNS 		: UINT := 2;
	MAX_CSV_FIELD_LENGTH	: UINT := 100;
END_VAR
VAR
	sNetId		: T_AmsNetId	:= ''; (* TwinCAT system network address *)
	sCSVLine	: T_MaxString	:= ''; (* Single CSV text line (row, record), we are using string as record buffer (your are able to see read fields)  *)
	sCSVField	: T_MaxString	:= ''; (* Single CSV field value (column, record field) *)
	bError		: BOOL;
	nErrId		: UDINT;
	nRow		: UDINT			:= 0; (* Row number (record) *)
	nColumn		: UDINT			:= 0; (* Column number (record field) *)
	hFile		: UINT			:= 0; (* File handle of the source file *)
	step		: DWORD			:= 0;
	fbFileOpen	: FB_FileOpen; (* Opens file *)
	fbFileClose	: FB_FileClose; (* Closes file *)
	fbFileGets	: FB_FileGets; (* Reads one record (line) *)
	fbReader	: FB_CSVMemBufferReader; (* Helper function block used to parse CSV data bytes (single record line) *)
END_VAR

// source: http://infosys.beckhoff.com/content/1033/tcplclibutilities/html/tcplclibutilities_csv_sample.htm 

DEFAULT_CSV_FIELD_SEP := 16#2C;(* Comma ASCII code *)
//DEFAULT_CSV_FIELD_SEP := 16#3B;(* Semicolon ASCII code *)

CASE step OF
	0:	(* Wait for rising edge at bRead variable *)
		IF bRead THEN
			bRead	:= FALSE;
			bBusy	:= TRUE;
			bError	:= FALSE;
			nErrId	:= 0;
			hFile	:= 0;
			nRow	:= 0;
			nColumn	:= 0;
			MEMSET( ADR( values ), 0, SIZEOF( values ) );
			step	:= 1;
		END_IF

	1:	(* Open source file *)
		fbFileOpen(bExecute := FALSE);
		fbFileOpen(sNetId := sNetId, sPathName := sFileName, nMode := FOPEN_MODEREAD OR FOPEN_MODETEXT, ePath := PATH_GENERIC, bExecute := TRUE);
		step := 2;

	2:(* Wait until open not busy *)
		fbFileOpen(bExecute := FALSE, bError => bError, nErrID => nErrID, hFile => hFile);
		IF NOT fbFileOpen.bBusy THEN
			IF NOT fbFileOpen.bError THEN
				step := 3;
			ELSE(* Error: file not found? *)
				step := 100;
			END_IF
		END_IF

	3:	(* Read single line (record) *)
		fbFileGets(bExecute := FALSE);
		fbFileGets(sNetId := sNetId, hFile := hFile, bExecute := TRUE);
		step := 4;

	4:(* Wait until read not busy *)
		fbFileGets(bExecute := FALSE, bError => bError, nErrID => nErrID, sLine => sCSVLine);
		IF NOT fbFileGets.bBusy THEN
			IF NOT fbFileGets.bError THEN
				IF fbFileGets.bEOF THEN
					step := 10;(* End of file reached => Close source file *)
				ELSE
					(* FB_FileGets returns text line without the CR (carriage return) character.
					We have to restore the CR character (replace the $L character with $R$L characters) *)
					IF Tc2_Standard.RIGHT( sCSVLine, 1 ) = '$L' THEN
						sCSVLine := REPLACE( sCSVLine, '$R$L', 2, LEN( sCSVLine ) );
					END_IF
					step := 5;
				END_IF
			ELSE(* Error *)
				step := 100;
			END_IF
		END_IF

	5:(* Parse single line (record) *)
		fbReader.eCmd := eEnumCmd_First; (* Read first field value *)
		REPEAT
			fbReader( pBuffer := ADR( sCSVLine ), cbBuffer := SIZEOF( sCSVLine ), getValue =>sCSVField );
			IF fbReader.bOk THEN
				fbReader.eCmd := eEnumCmd_Next; (* Read next field value *)

				IF (nRow < MAX_CSV_ROWS) THEN
					IF (nColumn < MAX_CSV_COLUMNS) THEN
						values[nRow, nColumn] := CSVFIELD_TO_STRING( sCSVField, FALSE );(* TODO: Save or use the field value in your application *)
						// remove ' ' from left side
						WHILE (Tc2_Standard.LEFT(values[nRow, nColumn], 1)=' ') DO
							values[nRow, nColumn] := Tc2_Standard.DELETE(values[nRow, nColumn],1,1);
						END_WHILE
						// remove ' ' from right side
						WHILE (Tc2_Standard.RIGHT(values[nRow, nColumn], 1)=' ') DO
							values[nRow, nColumn] := Tc2_Standard.DELETE(values[nRow, nColumn],1,LEN(values[nRow, nColumn]));
						END_WHILE
					END_IF
				END_IF

				nColumn := nColumn + 1; (* Increment number of read columns *)
				IF fbReader.bCRLF THEN (* CRLF == TRUE => End of reacord reached *)
					nRow 		:= nRow + 1; (* Increment number of read records *)
					nColumn 	:= 0; (* Reset number of columns *)
				END_IF

			ELSE (* Error: End of record reached or all fields read *)
				step := 3; (* Try to read next line *)
			END_IF
		UNTIL NOT fbReader.bOk
		END_REPEAT

	10:	(* Close source file *)
		fbFileClose(bExecute := FALSE);
		fbFileClose(sNetId := sNetId, hFile := hFile, bExecute := TRUE);
		step := 11;

	11:(* Wait until close not busy *)
		fbFileClose(bExecute := FALSE, bError => bError, nErrID => nErrID);
		IF (NOT fbFileClose.bBusy) THEN
			hFile := 0;
			step := 100;
		END_IF

	100: (* Error or ready step => cleanup *)
		IF (hFile <> 0) THEN
			step := 10; (* Close the source file *)
		ELSE
			bBusy := FALSE;
			step := 0; (* Ready *)
		END_IF

END_CASE

PROPERTY NumOfColumns : UINT
GET
NumOfColumns := MAX_CSV_COLUMNS;
END_GET
END_PROPERTY

PROPERTY NumOfRows : UINT
GET
NumOfRows := MAX_CSV_ROWS;
END_GET
END_PROPERTY

END_FUNCTION_BLOCK

// POUs/Utility/Data Channel/IdBase/FB_IdBaseRecvDch
FUNCTION_BLOCK FB_IdBaseRecvDch EXTENDS FB_DataChannelRecvBase IMPLEMENTS I_DataChannelRecv
VAR
	/// Saber Inteface Variables
	/// -----------------------------------------------------------------
	m_pInputData: POINTER TO T_IdBase_DCH;
END_VAR

SUPER^();

{attribute 'object_name' := 'GetData'}
METHOD GetData : BOOL
VAR_INPUT
	udiDataSize: UDINT;
	pData: POINTER TO BYTE;
END_VAR
GetData := FALSE;

IF m_eState = E_SaberPlcDHCState.DataReady THEN
	IF (udiDataSize > 0 ) AND (pData <> TC3_MEMMAN.NULL) THEN
		TC2_SYSTEM.MEMCPY(destAddr := pData, srcAddr := m_pInputData, n := udiDataSize);
		m_eState := E_SaberPlcDHCState.Acknowledge;	
		GetData := TRUE;
	END_IF	
END_IF
END_METHOD

{attribute 'object_name' := 'InitChannel'}
METHOD InitChannel : BOOL
VAR_INPUT
	udiDataSize: UDINT;
	pInputData: POINTER TO BYTE;
END_VAR
InitChannel := FALSE;

IF udiDataSize > 0 THEN
	IF pInputData <> TC3_MEMMAN.NULL THEN
		m_uinDataSize := udiDataSize;
		m_pInputData := pInputData;
		m_eState := E_SaberPlcDHCState.Init;
		InitChannel := TRUE;
	END_IF
END_IF
END_METHOD

END_FUNCTION_BLOCK

// POUs/Utility/DCH [Data Channel Base]/FB_DataChannelRecvBase
FUNCTION_BLOCK FB_DataChannelRecvBase IMPLEMENTS I_DataChannelRecv
VAR_INPUT
	pOutputDataBuffer: POINTER TO BYTE;
END_VAR
VAR CONSTANT
	cDataState_DONE: INT := -1;
	cDataState_Ready: INT := 1;
	cDataState_Retry: INT := -99;
	cDataState_Error: INT := -100;
	cMAX_RETRY: INT := 10;
END_VAR
VAR
	/// Saber Inteface Variables
	/// -----------------------------------------------------------------
	m_uinDataSize: UDINT;
	///	m_pInputData				: POINTER TO T_IdBase_DCH;
	m_iDchConfirm: INT;
	/// Local Variables
	/// -----------------------------------------------------------------
	m_eError: E_DCH_Error;
	m_eState: E_SaberPlcDHCState := E_SaberPlcDHCState.WaitChannelInit;
	m_intCountRetry: INT;
	m_iIdx: UDINT;
END_VAR

CASE m_eState OF
	E_SaberPlcDHCState.Init:
		m_intCountRetry := 0;
		m_eError := E_DCH_Error.None;
		m_iDchConfirm := cDataState_DONE;
		m_eState := E_SaberPlcDHCState.WaitForData;
		
	E_SaberPlcDHCState.WaitForData:
		IF m_iDchConfirm = cDataState_Ready THEN
			m_eState := E_SaberPlcDHCState.DataReady;
		END_IF

	E_SaberPlcDHCState.DataReady:
		; // The data can be retrieved
		
	E_SaberPlcDHCState.Acknowledge:
		// Delete all values

		// Acknowledge communication
		m_iDchConfirm := cDataState_DONE;
		m_eState := E_SaberPlcDHCState.WaitForData;
		
	E_SaberPlcDHCState.Retry:
		m_iDchConfirm := cDataState_Retry;
		m_eState := E_SaberPlcDHCState.WaitForData;

		m_eError := E_DCH_Error.Unknown;
	
END_CASE

PROPERTY Busy : BOOL
GET
Busy := m_eState <> E_SaberPlcDHCState.DataReady;
END_GET
END_PROPERTY

PROPERTY DataSize : UDINT
GET
DataSize := m_uinDataSize;
END_GET
END_PROPERTY

PROPERTY Error : INT
GET
Error := m_eError;
END_GET
SET
m_iDchConfirm := cDataState_Error;
m_eState := E_SaberPlcDHCState.Error;
END_SET
END_PROPERTY

{attribute 'object_name' := 'GetData'}
METHOD GetData : BOOL
VAR_INPUT
	udiDataSize: UDINT;
	pData: POINTER TO BYTE;
END_VAR
END_METHOD

{attribute 'object_name' := 'InitChannel'}
METHOD InitChannel : BOOL
VAR_INPUT
	udiDataSize: UDINT;
	pInputData: POINTER TO BYTE;
END_VAR
END_METHOD

END_FUNCTION_BLOCK

// POUs/Utility/DCH [Data Channel Base]/I_DataChannelRecv
INTERFACE I_DataChannelRecv

PROPERTY Busy : BOOL
GET
END_GET
END_PROPERTY

PROPERTY DataSize : UDINT
GET
END_GET
END_PROPERTY

PROPERTY Error : INT
GET
END_GET
SET
END_SET
END_PROPERTY

{attribute 'object_name' := 'GetData'}
METHOD GetData : BOOL
VAR_INPUT
	udiDataSize: UDINT;
	pData: POINTER TO BYTE;
END_VAR
END_METHOD

{attribute 'object_name' := 'InitChannel'}
METHOD InitChannel : BOOL
VAR_INPUT
	udiDataSize: UDINT;
	pInputData: POINTER TO BYTE;
END_VAR
END_METHOD

END_INTERFACE

// POUs/Utility/Data Channel/IdBase/FB_IdBaseSendDch
FUNCTION_BLOCK FB_IdBaseSendDch EXTENDS FB_DataChannelSendBase IMPLEMENTS I_DataChannelSend
VAR
	/// Saber Inteface Variables
	/// -----------------------------------------------------------------
	m_pOutputData: POINTER TO T_IdBase_DCH;
END_VAR

SUPER^();

{attribute 'object_name' := 'InitChannel'}
METHOD InitChannel : BOOL
VAR_INPUT
	udiDataSize: UDINT;
	pOutputData: POINTER TO BYTE;
END_VAR
InitChannel := FALSE;

IF udiDataSize > 0 THEN
	IF pOutputData <> TC3_MEMMAN.NULL THEN
		m_uinDataSize := udiDataSize;
		m_pOutputData := pOutputData;
		m_eState := E_PlcSaberDHCState.Init;
		InitChannel := TRUE;
	END_IF
END_IF
END_METHOD

{attribute 'object_name' := 'SendData'}
METHOD SendData : BOOL
VAR_INPUT
	udiDataSize: UDINT;
	pData: POINTER TO BYTE;
END_VAR
SendData := FALSE;

IF m_eState = E_PlcSaberDHCState.WaitForJob THEN
	IF (udiDataSize > 0 ) AND (pData <> TC3_MEMMAN.NULL) THEN
		TC2_SYSTEM.MEMCPY(destAddr := m_pOutputData, srcAddr := pData, n := udiDataSize);
		m_eState := E_PlcSaberDHCState.SendData;	
		SendData := TRUE;
	END_IF	
END_IF
END_METHOD

END_FUNCTION_BLOCK

// POUs/Utility/DCH [Data Channel Base]/FB_DataChannelSendBase
FUNCTION_BLOCK FB_DataChannelSendBase IMPLEMENTS I_DataChannelSend
VAR CONSTANT
	cMAX_DATACHANNEL_ITEM_SIZE: UINT := 200;
	cMAX_RETRY: INT := 10;
	cDataState_DONE: INT := -1;
	cDataCmd_Ready: INT := 1;
	cDataCmd_ClearBuffer: INT := -98;
	cDataCmd_Retry: INT := -99;
	cDataCmd_Error: INT := -100;
END_VAR
VAR
	/// Saber Inteface Variables
	/// -----------------------------------------------------------------
	m_uinDataSize: UDINT;
	///	m_pOutputData				: POINTER TO T_IdBase_DCH;
	m_iDchConfirm: INT;
	/// Local Variables
	/// -----------------------------------------------------------------
	m_eState: E_PlcSaberDHCState := E_PlcSaberDHCState.Init;
	m_eError: E_DCH_Error;
	m_intCountRetry: INT;
END_VAR

CASE m_eState OF
	E_PlcSaberDHCState.Init:
		m_eError := E_DCH_Error.None;
		m_eState := E_PlcSaberDHCState.WaitForJob;
		m_iDchConfirm := cDataState_DONE;
		
	E_PlcSaberDHCState.WaitForJob:
		;  // Method SendData is needed to go out of this state
		
	E_PlcSaberDHCState.SendData:
		m_iDchConfirm := cDataCmd_Ready;
		m_eState := E_PlcSaberDHCState.Acknowledge;
		
	E_PlcSaberDHCState.Acknowledge:
		CASE m_iDchConfirm OF
			cDataState_DONE:
				m_iDchConfirm := cDataState_DONE;
				m_eState := E_PlcSaberDHCState.WaitForJob;
			cDataCmd_Retry:
				m_eState := E_PlcSaberDHCState.Retry;
			cDataCmd_Error:	
				m_eState := E_PlcSaberDHCState.Error;
			cDataCmd_ClearBuffer:	
				m_eState := E_PlcSaberDHCState.ClearBufferBusy;
		END_CASE
		
	E_PlcSaberDHCState.Retry:
		IF m_intCountRetry < cMAX_RETRY THEN
			m_intCountRetry := m_intCountRetry + 1;
			m_eState := E_PlcSaberDHCState.SendData;
		ELSE
			m_eState := E_PlcSaberDHCState.Error;
		END_IF
		
	E_PlcSaberDHCState.Error:
		m_eError := E_DCH_Error.Unknown;
		m_eState := E_PlcSaberDHCState.WaitForJob;

	E_PlcSaberDHCState.ClearBufferBusy:
		// Wait for method ClearBufferDone call

	E_PlcSaberDHCState.ClearBufferDone:
		m_iDchConfirm := cDataState_DONE;
		m_eState := E_PlcSaberDHCState.WaitForJob;
END_CASE

PROPERTY Busy : BOOL
GET
Busy := m_eState <> E_PlcSaberDHCState.WaitForJob;
END_GET
END_PROPERTY

{attribute 'object_name' := 'ClearBufferDone'}
METHOD ClearBufferDone : BOOL
m_eState := E_PlcSaberDHCState.ClearBufferDone;
END_METHOD

PROPERTY ClearBufferRequest : BOOL
GET
ClearBufferRequest := m_eState = E_PlcSaberDHCState.ClearBufferBusy;
END_GET
END_PROPERTY

PROPERTY DataSize : UDINT
GET
DataSize := m_uinDataSize;
END_GET
END_PROPERTY

PROPERTY Error : INT
GET
Error := m_eError;
END_GET
SET
END_SET
END_PROPERTY

{attribute 'object_name' := 'InitChannel'}
METHOD InitChannel : BOOL
VAR_INPUT
	udiDataSize: UDINT;
	pOutputData: POINTER TO BYTE;
END_VAR
END_METHOD

{attribute 'object_name' := 'SendData'}
METHOD SendData : BOOL
VAR_INPUT
	udiDataSize: UDINT;
	pData: POINTER TO BYTE;
END_VAR
END_METHOD

END_FUNCTION_BLOCK

// POUs/Utility/DCH [Data Channel Base]/I_DataChannelSend
INTERFACE I_DataChannelSend

PROPERTY Busy : BOOL
GET
END_GET
END_PROPERTY

{attribute 'object_name' := 'ClearBufferDone'}
METHOD ClearBufferDone : BOOL
END_METHOD

PROPERTY ClearBufferRequest : BOOL
GET
END_GET
END_PROPERTY

PROPERTY DataSize : UDINT
GET
END_GET
END_PROPERTY

PROPERTY Error : INT
GET
END_GET
SET
END_SET
END_PROPERTY

{attribute 'object_name' := 'InitChannel'}
METHOD InitChannel : BOOL
VAR_INPUT
	udiDataSize: UDINT;
	pOutputData: POINTER TO BYTE;
END_VAR
END_METHOD

{attribute 'object_name' := 'SendData'}
METHOD SendData : BOOL
VAR_INPUT
	udiDataSize: UDINT;
	pData: POINTER TO BYTE;
END_VAR
END_METHOD

END_INTERFACE

// POUs/Utility/DCH [Data Channel Base]/FB_DataChannelRecvFifo
FUNCTION_BLOCK FB_DataChannelRecvFifo EXTENDS FB_ArrayFifo
VAR
	m_pDataChannel: POINTER TO FB_DataChannelRecvBase;
	m_bolEnable: BOOL;
	m_intMaxFifoSize: INT := 10;
	m_pItem: POINTER TO BYTE;
	m_bolResult: BOOL;
END_VAR

IF m_bolEnable AND (m_pItem <> Tc3_MemMan.NULL) THEN
	IF NOT m_pDataChannel^.Busy THEN
		m_bolResult := m_pDataChannel^.GetData(
						udiDataSize := m_pDataChannel^.DataSize,
						pData		:= m_pItem);

		IF m_uinItemCount < m_uinMaxItemCount THEN
			Push(m_pItem);
		ELSE
			m_pDataChannel^.Error := 1;
		END_IF 	
	END_IF
	
	m_pDataChannel^();
END_IF

PROPERTY DataChannel : POINTER TO FB_DataChannelRecvBase
SET
m_pDataChannel := DataChannel;
END_SET
END_PROPERTY

PROPERTY Enable : BOOL
GET
Enable := m_bolEnable;
END_GET
SET
m_bolEnable := Enable;
END_SET
END_PROPERTY

PROPERTY Item : POINTER TO BYTE
GET
END_GET
SET
m_pItem := Item;
END_SET
END_PROPERTY

PROPERTY MaxFifoSize : INT
GET
MaxFifoSize := m_intMaxFifoSize;
END_GET
SET
m_intMaxFifoSize := MaxFifoSize;
END_SET
END_PROPERTY

END_FUNCTION_BLOCK

// POUs/Utility/DCH [Data Channel Base]/FB_DataChannelSenderFifo
FUNCTION_BLOCK FB_DataChannelSenderFifo EXTENDS FB_DynamicFifo
VAR
	m_pDataChannel: POINTER TO FB_DataChannelSendBase;
	m_pItem: POINTER TO BYTE;
	m_bolEnable: BOOL;
	m_intMaxFifoSize: INT := 10;
	bResult: BOOL;
END_VAR

IF (m_uinItemCount > 0) AND NOT m_pDataChannel^.Busy THEN
	m_pItem := Pop();

	IF m_bolEnable THEN
		bResult := m_pDataChannel^.SendData(
						pData       := m_pItem,
						udiDataSize := m_pDataChannel^.DataSize);
	END_IF;
	
	IF m_bFreeDataPointer THEN
		__DELETE(m_pItem);
	END_IF
END_IF

IF m_pDataChannel^.ClearBufferRequest THEN
	THIS^.ClearFifo();
	m_pDataChannel^.ClearBufferDone();
END_IF

m_pDataChannel^();

PROPERTY DataChannel : POINTER TO FB_DataChannelSendBase
SET
m_pDataChannel := DataChannel;
END_SET
END_PROPERTY

PROPERTY Enable : BOOL
GET
Enable := m_bolEnable;
END_GET
SET
IF m_bolEnable AND NOT Enable THEN
	THIS^.ClearFifo();
END_IF

m_bolEnable := Enable;
END_SET
END_PROPERTY

PROPERTY MaxFifoSize : INT
GET
MaxFifoSize := m_intMaxFifoSize;
END_GET
SET
m_intMaxFifoSize := MaxFifoSize;
END_SET
END_PROPERTY

END_FUNCTION_BLOCK

// POUs/Utility/DFF [Dynamic Pointer FiFo]/FB_DynamicFifo
FUNCTION_BLOCK FB_DynamicFifo
VAR
	/// Configuration
	m_bFreeDataPointer: BOOL;
	/// Actual Count of the elements in the buffer
	m_uinItemCount: UINT;
	/// Index of the first added element
	m_pFirstElement: POINTER TO T_QueueBase;
	/// Index of the last added element
	m_pLastElement: POINTER TO T_QueueBase;
END_VAR

{attribute 'object_name' := 'ClearFifo'}
METHOD ClearFifo : BOOL
VAR
	pItem: POINTER TO T_QueueBase;
	pNextItem: POINTER TO T_QueueBase;
END_VAR
pItem := m_pFirstElement;
m_pFirstElement := NULL;

WHILE pItem <> TC3_MEMMAN.NULL DO
	pNextItem := pItem^.pNext;
	
	IF m_bFreeDataPointer THEN
		__DELETE(pItem^.pData);
	END_IF
	
	__DELETE(pItem);
	pItem := pNextItem;
END_WHILE

m_pLastElement := NULL;
m_uinItemCount := 0;
END_METHOD

PROPERTY FreeDataPointer : BOOL
GET
FreeDataPointer := m_bFreeDataPointer;
END_GET
SET
m_bFreeDataPointer := FreeDataPointer;
END_SET
END_PROPERTY

PROPERTY ItemCount : UINT
GET
ItemCount := m_uinItemCount;
END_GET
END_PROPERTY

{attribute 'object_name' := 'Peek'}
METHOD Peek : POINTER TO BYTE
Peek := TC3_MEMMAN.NULL;

IF m_uinItemCount > 0 THEN
	Peek := m_pFirstElement^.pData;
END_IF
END_METHOD

{attribute 'object_name' := 'Pop'}
METHOD Pop : POINTER TO BYTE
VAR
	pItem: POINTER TO T_QueueBase;
END_VAR
Pop := TC3_MEMMAN.NULL;

IF m_uinItemCount > 0 THEN
	pItem := m_pFirstElement;
	
	m_pFirstElement := m_pFirstElement^.pNext;

	IF m_pFirstElement <> TC3_MEMMAN.NULL THEN
		m_pFirstElement^.pPrevious := TC3_MEMMAN.NULL;
	ELSE
		m_pLastElement := TC3_MEMMAN.NULL;
	END_IF

	m_uinItemCount := m_uinItemCount - 1;

	Pop := pItem^.pData;
	__DELETE(pItem);
END_IF
END_METHOD

{attribute 'object_name' := 'Push'}
METHOD Push : INT
VAR_INPUT
	pData: POINTER TO BYTE;
END_VAR
VAR
	pItem: POINTER TO T_QueueBase;
END_VAR
pItem := __NEW(T_QueueBase);
pItem^.pData := pData;

IF m_uinItemCount = 0 THEN
	m_pFirstElement := pItem;
	m_pLastElement  := pItem;
	pItem^.pNext := TC3_MEMMAN.NULL;
	pItem^.pPrevious := TC3_MEMMAN.NULL;
ELSE
	m_pLastElement^.pNext:= pItem;
	pItem^.pPrevious := m_pLastElement;
	pItem^.pNext := TC3_MEMMAN.NULL;
	m_pLastElement  := pItem;
END_IF

m_uinItemCount := m_uinItemCount + 1;

Push := UINT_TO_INT(m_uinItemCount);
END_METHOD

END_FUNCTION_BLOCK

// POUs/Utility/GHT [Generic Hash Table]/FB_GHT
FUNCTION_BLOCK FB_GHT IMPLEMENTS IGHT
VAR CONSTANT
	MAX_HASH_LISTS: INT := 3;
	MAX_HASHLIST_ENTRIES: INT := 50;
	CUTOFF_A: ULINT := 4000000000;
	CUTOFF_B: ULINT := 8000000000;
END_VAR
VAR
	m_bolDeleteItems: BOOL;
	m_uintCount: UINT;
	m_fbHashTable: ARRAY[0..(MAX_HASH_LISTS - 1)] OF FB_HashTableCtrl;
	m_hHashTable: ARRAY[0..(MAX_HASH_LISTS - 1)] OF T_HHASHTABLE;
	m_uliCutoff: ARRAY[0..(MAX_HASH_LISTS - 1)] OF ULINT;
	m_aHashTableBuffer: ARRAY[0..(MAX_HASH_LISTS - 1)] OF T_GHTHashTableBuffer;
END_VAR

{attribute 'object_name' := 'AddItem'}
METHOD AddItem : BOOL
VAR_INPUT
	uliKey: ULINT;
	pData: POINTER TO BYTE;
END_VAR
VAR
	iIdx: INT;
END_VAR
iIdx := GetTableIdx(uliKey);

m_fbHashTable[iIdx].A_Add( key := ULINT_TO_UDINT(uliKey-m_uliCutoff[iIdx]), putValue := pData, hTable := m_hHashTable[iIdx] );

IF m_fbHashTable[iIdx].bOk THEN
	m_uintCount := m_uintCount + 1;
END_IF
END_METHOD

{attribute 'object_name' := 'Clear'}
METHOD Clear : BOOL
VAR_INPUT
	bolFreePointer: BOOL;
END_VAR
VAR
	iIdx: INT;
	pData: POINTER TO BYTE;
END_VAR
FOR iIdx := 0 TO MAX_HASH_LISTS - 1 DO
	IF bolFreePointer THEN
		m_fbHashTable[iIdx].A_GetFirst(hTable := m_hHashTable[iIdx]);

		WHILE m_fbHashTable[iIdx].bOk DO
			pData := m_fbHashTable[iIdx].getValue;
			__DELETE(pData);
			m_fbHashTable[iIdx].A_GetNext(hTable := m_hHashTable[iIdx]);
		END_WHILE
		
	END_IF
	
	m_fbHashTable[iIdx].A_RemoveAll(hTable := m_hHashTable[iIdx]);
END_FOR

m_uintCount := 0;
END_METHOD

PROPERTY Count : UINT
GET
END_GET
END_PROPERTY

{attribute 'object_name' := 'FB_init'}
METHOD FB_init : BOOL
VAR_INPUT
	/// if TRUE, the retain variables are initialized (warm start / cold start)
	bInitRetains: BOOL;
	/// if TRUE, the instance afterwards gets moved into the copy code (online change)
	bInCopyCode: BOOL;
END_VAR
m_uliCutoff[0] := 0;
m_uliCutoff[1] := CUTOFF_A;
m_uliCutoff[2] := CUTOFF_B;

m_uintCount := 0;
END_METHOD

{attribute 'object_name' := 'GetTableIdx'}
METHOD PRIVATE GetTableIdx : INT
VAR_INPUT
	uliBarcode: ULINT;
END_VAR
IF uliBarcode < CUTOFF_A THEN
	GetTableIdx := 0;
	RETURN;
END_IF

IF uliBarcode > CUTOFF_B THEN
	GetTableIdx := 2;
	RETURN;
END_IF

GetTableIdx := 1;
END_METHOD

{attribute 'object_name' := 'Initialize'}
METHOD Initialize : BOOL
F_CreateHashTableHnd( ADR( m_aHashTableBuffer[0].aBuffer ), SIZEOF( m_aHashTableBuffer[0].aBuffer ), m_hHashTable[0] );
F_CreateHashTableHnd( ADR( m_aHashTableBuffer[1].aBuffer ), SIZEOF( m_aHashTableBuffer[1].aBuffer ), m_hHashTable[1] );
F_CreateHashTableHnd( ADR( m_aHashTableBuffer[2].aBuffer ), SIZEOF( m_aHashTableBuffer[2].aBuffer ), m_hHashTable[2] );
END_METHOD

{attribute 'object_name' := 'Lookup'}
METHOD Lookup : POINTER TO BYTE
VAR_INPUT
	uliKey: ULINT;
	bolRemove: BOOL;
END_VAR
VAR
	pfbHashTable: POINTER TO FB_HashTableCtrl;
	phHashTable: POINTER TO T_HHASHTABLE;
	uliCutoff: ULINT;
	iIdx: INT;
END_VAR
iIdx := GetTableIdx(uliKey);

m_fbHashTable[iIdx].A_Lookup( key := ULINT_TO_UDINT(uliKey-m_uliCutoff[iIdx]), hTable := m_hHashTable[iIdx] );

IF m_fbHashTable[iIdx].bOk THEN
	Lookup := m_fbHashTable[iIdx].getValue;
	
	IF bolRemove THEN
		m_fbHashTable[iIdx].A_Remove( key := ULINT_TO_UDINT(uliKey-m_uliCutoff[iIdx]), hTable := m_hHashTable[iIdx]);

		IF m_fbHashTable[iIdx].bOk THEN
			m_uintCount := m_uintCount - 1;
		END_IF
	END_IF
ELSE
	Lookup := NULL;
END_IF
END_METHOD

END_FUNCTION_BLOCK

// POUs/Utility/GHT [Generic Hash Table]/IGHT
INTERFACE IGHT

{attribute 'object_name' := 'AddItem'}
METHOD AddItem : BOOL
VAR_INPUT
	uliKey: ULINT;
	pData: POINTER TO BYTE;
END_VAR
END_METHOD

{attribute 'object_name' := 'Clear'}
METHOD Clear : BOOL
VAR_INPUT
	bolFreePointer: BOOL;
END_VAR
END_METHOD

PROPERTY Count : UINT
GET
END_GET
END_PROPERTY

{attribute 'object_name' := 'Initialize'}
METHOD Initialize : BOOL
END_METHOD

{attribute 'object_name' := 'Lookup'}
METHOD Lookup : POINTER TO BYTE
VAR_INPUT
	uliKey: ULINT;
	bolRemove: BOOL;
END_VAR
END_METHOD

END_INTERFACE
